// Mitsubishi GX Works2 project: RMUTI-QRCode_modbus   PLC: FX3U/FX3UC

PROGRAM MAIN
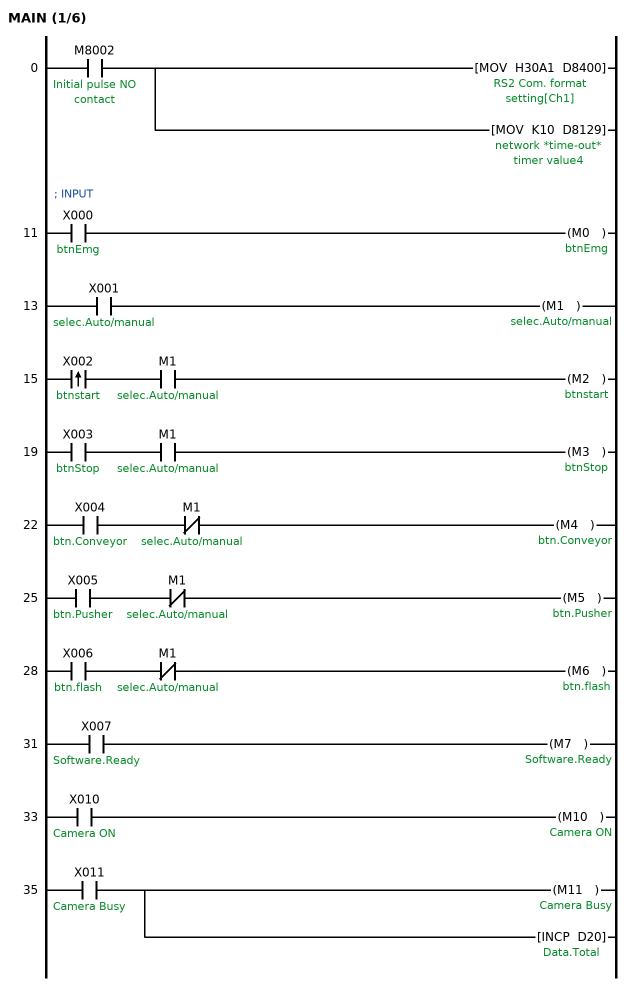
0     LD      M8002  ; Initial pulse NO contact
      MOV     H30A1 D8400  ; RS2 Com. format setting[Ch1]
      MOV     K10 D8129  ; network *time-out* timer value4
; INPUT
11    LD      X000  ; btnEmg
      OUT     M0  ; btnEmg
13    LD      X001  ; selec.Auto/manual
      OUT     M1  ; selec.Auto/manual
15    LDP     X002  ; btnstart
      AND     M1  ; selec.Auto/manual
      OUT     M2  ; btnstart
19    LD      X003  ; btnStop
      AND     M1  ; selec.Auto/manual
      OUT     M3  ; btnStop
22    LD      X004  ; btn.Conveyor
      ANI     M1  ; selec.Auto/manual
      OUT     M4  ; btn.Conveyor
25    LD      X005  ; btn.Pusher
      ANI     M1  ; selec.Auto/manual
      OUT     M5  ; btn.Pusher
28    LD      X006  ; btn.flash
      ANI     M1  ; selec.Auto/manual
      OUT     M6  ; btn.flash
31    LD      X007  ; Software.Ready
      OUT     M7  ; Software.Ready
33    LD      X010  ; Camera ON
      OUT     M10  ; Camera ON
35    LD      X011  ; Camera Busy
      OUT     M11  ; Camera Busy
      INCP    D20  ; Data.Total
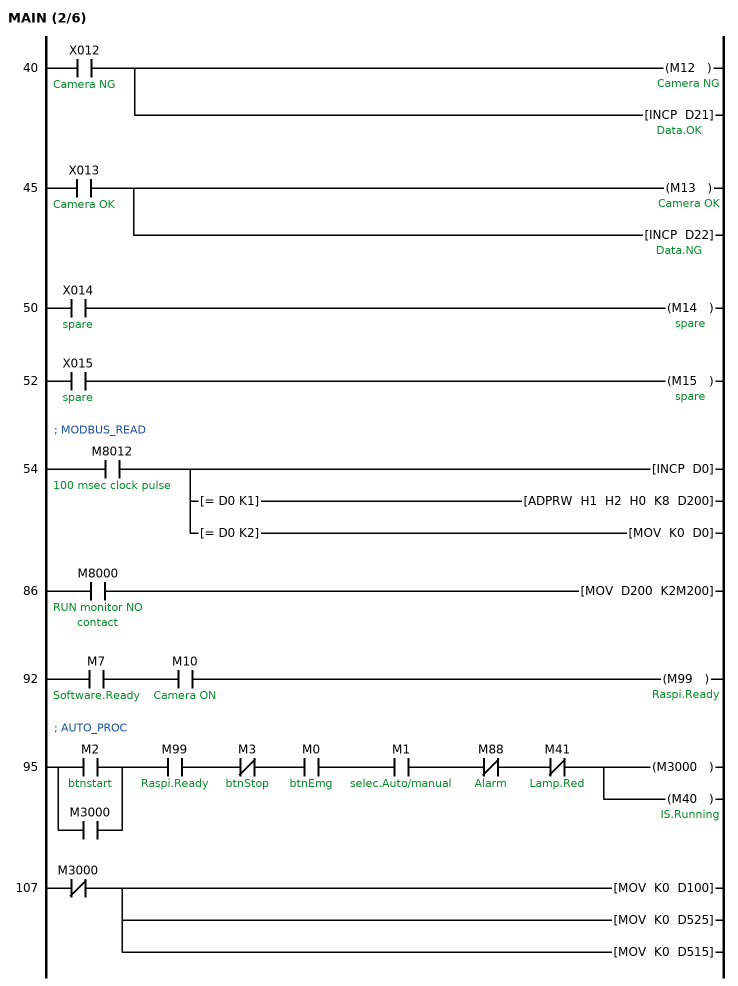
40    LD      X012  ; Camera NG
      OUT     M12  ; Camera NG
      INCP    D21  ; Data.OK
45    LD      X013  ; Camera OK
      OUT     M13  ; Camera OK
      INCP    D22  ; Data.NG
50    LD      X014  ; spare
      OUT     M14  ; spare
52    LD      X015  ; spare
      OUT     M15  ; spare
; MODBUS_READ
54    LD      M8012  ; 100 msec clock pulse
      INCP    D0
      MPS
      AND=    D0 K1
      ADPRW   H1 H2 H0 K8 D200
      MPP
      AND=    D0 K2
      MOV     K0 D0
86    LD      M8000  ; RUN monitor NO contact
      MOV     D200 K2M200  ; Sensor.IN
92    LD      M7  ; Software.Ready
      AND     M10  ; Camera ON
      OUT     M99  ; Raspi.Ready
; AUTO_PROC
95    LD      M2  ; btnstart
      OR      M3000
      AND     M99  ; Raspi.Ready
      ANI     M3  ; btnStop
      AND     M0  ; btnEmg
      AND     M1  ; selec.Auto/manual
      ANI     M88  ; Alarm
      ANI     M41  ; Lamp.Red
      OUT     M3000
      OUT     M40  ; IS.Running
107   LDI     M3000
      MOV     K0 D100
      MOV     K0 D525
      MOV     K0 D515
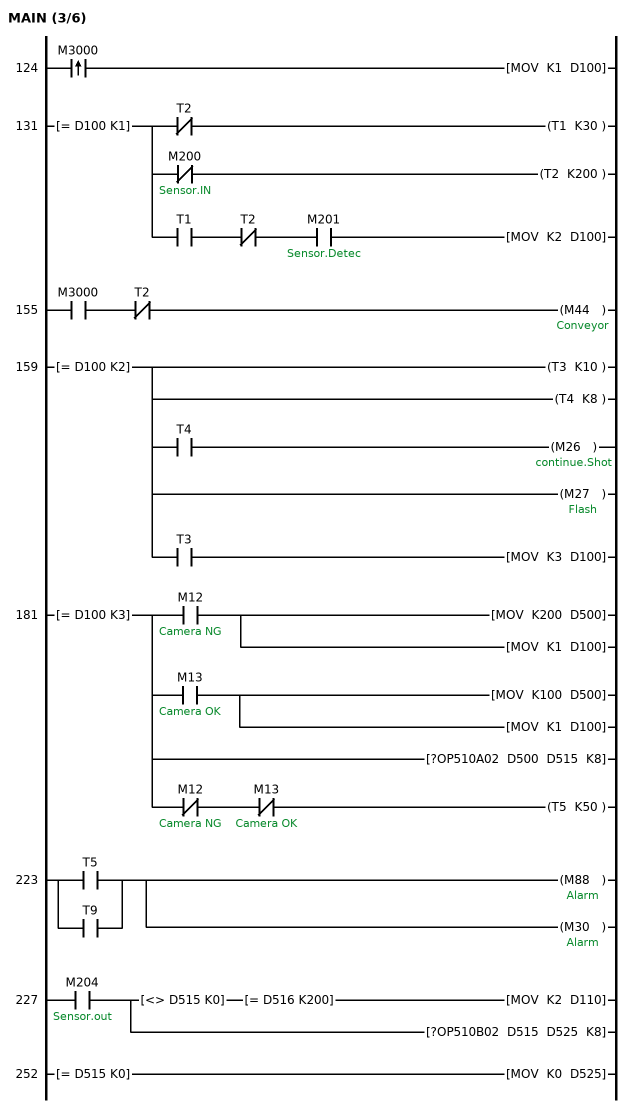
124   LDP     M3000
      MOV     K1 D100
131   LD=     D100 K1
      MPS
      ANI     T2
      OUT     T1 K30
      MRD
      ANI     M200  ; Sensor.IN
      OUT     T2 K200
      MPP
      AND     T1
      ANI     T2
      AND     M201  ; Sensor.Detec
      MOV     K2 D100
155   LD      M3000
      ANI     T2
      OUT     M44  ; Conveyor
159   LD=     D100 K2
      OUT     T3 K10
      OUT     T4 K8
      MPS
      AND     T4
      OUT     M26  ; continue.Shot
      MPP
      OUT     M27  ; Flash
      AND     T3
      MOV     K3 D100
181   LD=     D100 K3
      MPS
      AND     M12  ; Camera NG
      MOV     K200 D500
      MOV     K1 D100
      MRD
      AND     M13  ; Camera OK
      MOV     K100 D500
      MOV     K1 D100
      MPP
      ?OP510A02 D500 D515 K8
      ANI     M12  ; Camera NG
      ANI     M13  ; Camera OK
      OUT     T5 K50
223   LD      T5
      OR      T9
      OUT     M88  ; Alarm
      OUT     M30  ; Alarm
227   LD      M204  ; Sensor.out
      MPS
      AND<>   D515 K0
      AND=    D516 K200
      MOV     K2 D110
      MPP
      ?OP510B02 D515 D525 K8
252   LD=     D515 K0
      MOV     K0 D525
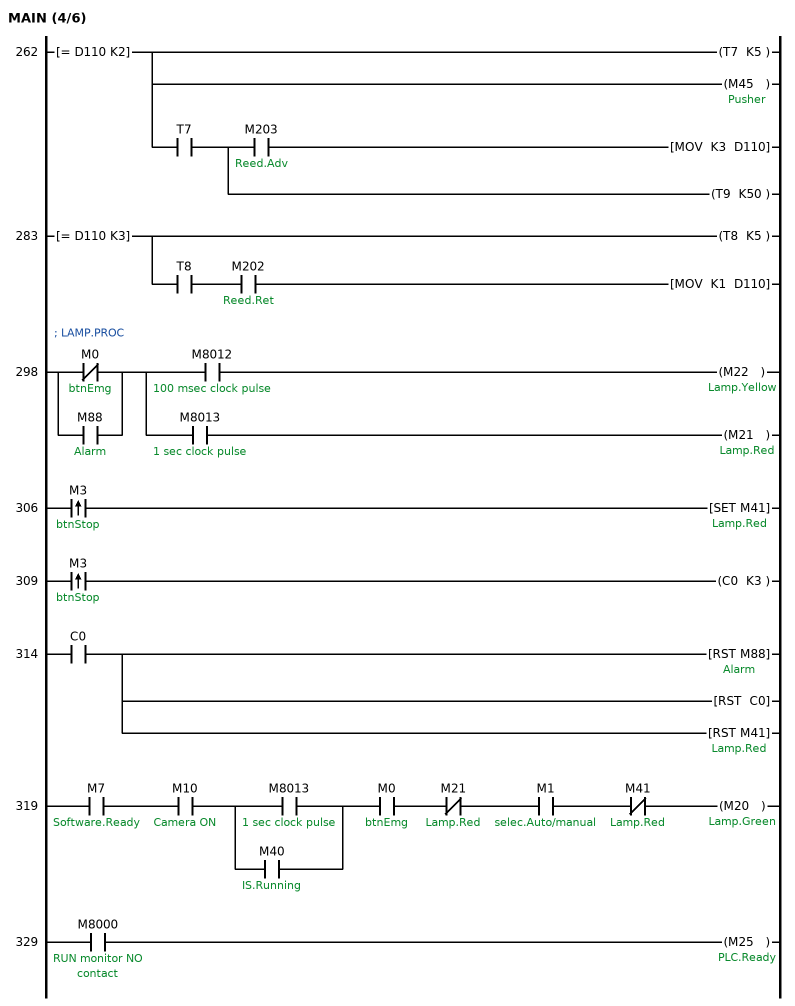
262   LD=     D110 K2
      OUT     T7 K5
      OUT     M45  ; Pusher
      AND     T7
      MPS
      AND     M203  ; Reed.Adv
      MOV     K3 D110
      MPP
      OUT     T9 K50
283   LD=     D110 K3
      OUT     T8 K5
      AND     T8
      AND     M202  ; Reed.Ret
      MOV     K1 D110
; LAMP.PROC
298   LDI     M0  ; btnEmg
      OR      M88  ; Alarm
      MPS
      AND     M8012  ; 100 msec clock pulse
      OUT     M22  ; Lamp.Yellow
      MPP
      AND     M8013  ; 1 sec clock pulse
      OUT     M21  ; Lamp.Red
306   LDP     M3  ; btnStop
      SET     M41  ; Lamp.Red
309   LDP     M3  ; btnStop
      OUT     C0 K3
314   LD      C0
      RST     M88  ; Alarm
      RST     C0
      RST     M41  ; Lamp.Red
319   LD      M7  ; Software.Ready
      AND     M10  ; Camera ON
      LD      M8013  ; 1 sec clock pulse
      OR      M40  ; IS.Running
      ANB
      AND     M0  ; btnEmg
      ANI     M21  ; Lamp.Red
      AND     M1  ; selec.Auto/manual
      ANI     M41  ; Lamp.Red
      OUT     M20  ; Lamp.Green
329   LD      M8000  ; RUN monitor NO contact
      OUT     M25  ; PLC.Ready
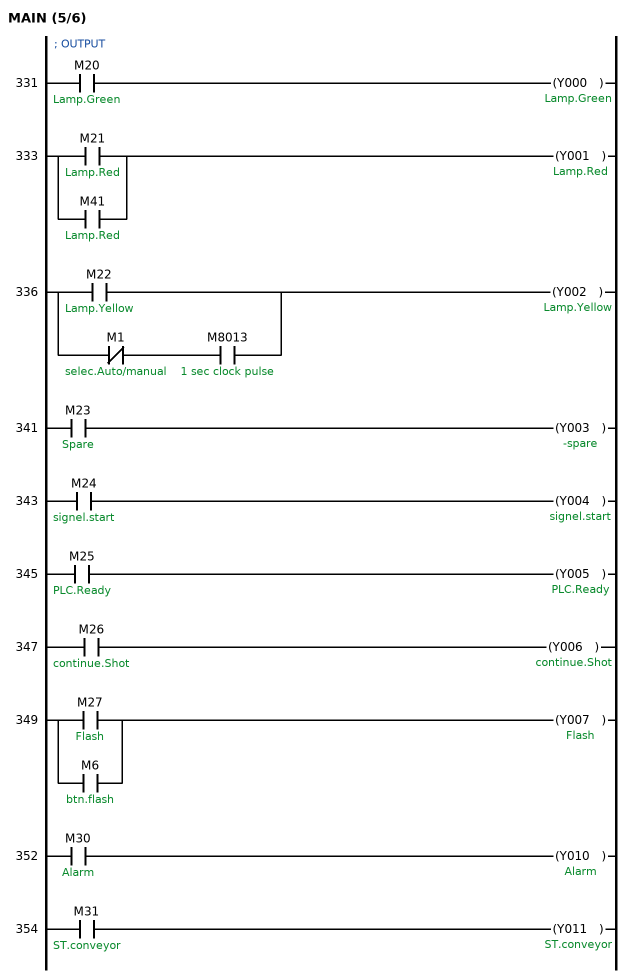
; OUTPUT
331   LD      M20  ; Lamp.Green
      OUT     Y000  ; Lamp.Green
333   LD      M21  ; Lamp.Red
      OR      M41  ; Lamp.Red
      OUT     Y001  ; Lamp.Red
336   LD      M22  ; Lamp.Yellow
      LDI     M1  ; selec.Auto/manual
      AND     M8013  ; 1 sec clock pulse
      ORB
      OUT     Y002  ; Lamp.Yellow
341   LD      M23  ; Spare
      OUT     Y003  ; -spare
343   LD      M24  ; signel.start
      OUT     Y004  ; signel.start
345   LD      M25  ; PLC.Ready
      OUT     Y005  ; PLC.Ready
347   LD      M26  ; continue.Shot
      OUT     Y006  ; continue.Shot
349   LD      M27  ; Flash
      OR      M6  ; btn.flash
      OUT     Y007  ; Flash
352   LD      M30  ; Alarm
      OUT     Y010  ; Alarm
354   LD      M31  ; ST.conveyor
      OUT     Y011  ; ST.conveyor
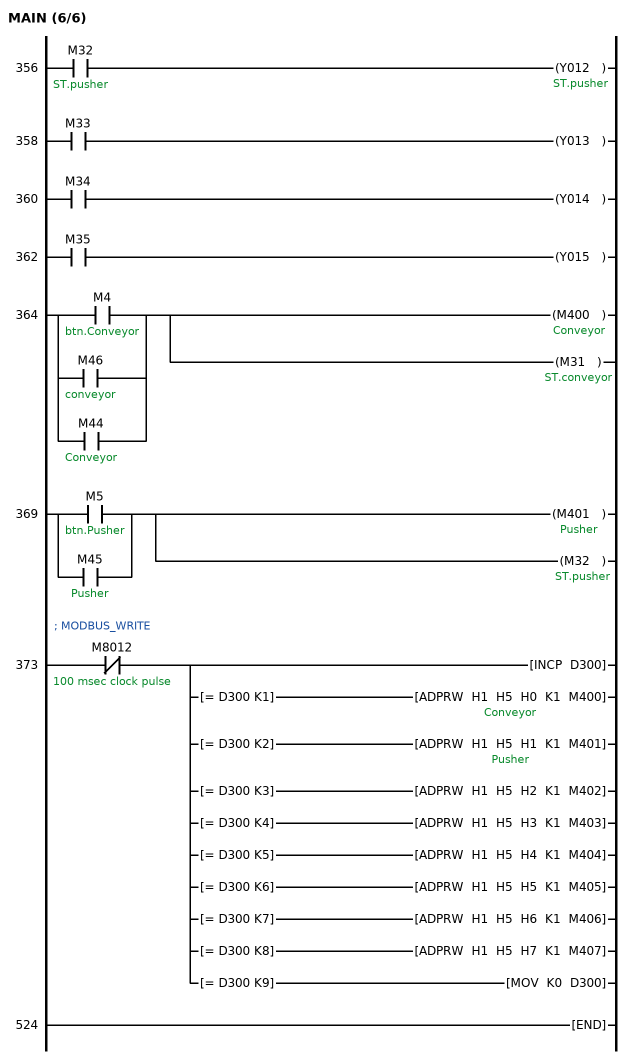
356   LD      M32  ; ST.pusher
      OUT     Y012  ; ST.pusher
358   LD      M33
      OUT     Y013
360   LD      M34
      OUT     Y014
362   LD      M35
      OUT     Y015
364   LD      M4  ; btn.Conveyor
      OR      M46  ; conveyor
      OR      M44  ; Conveyor
      OUT     M400  ; Conveyor
      OUT     M31  ; ST.conveyor
369   LD      M5  ; btn.Pusher
      OR      M45  ; Pusher
      OUT     M401  ; Pusher
      OUT     M32  ; ST.pusher
; MODBUS_WRITE
373   LDI     M8012  ; 100 msec clock pulse
      INCP    D300
      MPS
      AND=    D300 K1
      ADPRW   H1 H5 H0 K1 M400
      MRD
      AND=    D300 K2
      ADPRW   H1 H5 H1 K1 M401
      MRD
      AND=    D300 K3
      ADPRW   H1 H5 H2 K1 M402
      MRD
      AND=    D300 K4
      ADPRW   H1 H5 H3 K1 M403
      MRD
      AND=    D300 K5
      ADPRW   H1 H5 H4 K1 M404
      MRD
      AND=    D300 K6
      ADPRW   H1 H5 H5 K1 M405
      MRD
      AND=    D300 K7
      ADPRW   H1 H5 H6 K1 M406
      MRD
      AND=    D300 K8
      ADPRW   H1 H5 H7 K1 M407
      MPP
      AND=    D300 K9
      MOV     K0 D300
524   END
END_PROGRAM

// device comments not shown above
M16  ; Reed.Ret
M17  ; Reed.Adv
M18  ; Sensor
